// TIA Portal V15.1 export
// export: Created 2024-05-17T05:38:26.0543023Z, ExportSetting WithDefaults, DisplayName Totally Integrated Automation Portal, DisplayVersion V15.1 Update 5, DisplayName TIA Portal Openness, DisplayVersion V15.1 Update 5, DisplayName SINAMICS Startdrive Advanced, DisplayVersion V15.1, DisplayName G130, G150, S120, S150, SINAMICS MV, S210, DisplayVersion V15.1, DisplayName G110M, G120, G120C, G120D, G120P, DisplayVersion V15.1, DisplayName STEP 7 Professional, DisplayVersion V15.1 Update 5, DisplayName STEP 7 Safety, DisplayVersion V15.1, DisplayName WinCC Professional, DisplayVersion V15.1 Update 5, DisplayName SIMATIC Visualization Architect, DisplayVersion V15.1
FUNCTION "LETAFuseName" : Void   // FC2102, SCL
{ S7_Optimized_Access := 'TRUE' }
VERSION : 0.1
// stored: AutoNumber false, IsIECCheckEnabled false, SetENOAutomatically False, UDAEnableTagReadback false
   VAR_INPUT
      I_DBName : String;   // DB Name
      C_Config : "ETAFuseCPC20PNConfig";   // Config / Description About Type Of Object
   END_VAR
   VAR_OUTPUT
      O_FuseNr : Int;   // Fuse number in "STRUCT"
      O_FuseNameOK : Bool;   // Fuse name is found one time by the config
      O_FuseNameNOK : Bool;   // Fuse name is not found by the config or Instance name DB is wrong
      O_FuseNameMoreThenOne : Bool;   // Fuse name is found more then one time by the config
   END_VAR
   VAR_TEMP
      Index : Int;   // Index
      SubIndex : Int;   // Sub Index
   END_VAR
BEGIN
   #Index := 1;
   #SubIndex := 0;

   WHILE (#Index <= 64) DO
       IF (#C_Config.Fuse[#Index].Name = #I_DBName) THEN
           #O_FuseNr := #Index;
           #SubIndex := #SubIndex + 1;
       END_IF;
       #Index := #Index + 1;
   END_WHILE;

   IF (#SubIndex = 1) THEN
       #O_FuseNameOK := True;
       #O_FuseNameNOK := False;
       #O_FuseNameMoreThenOne := False;
   END_IF;

   IF (#SubIndex = 0) THEN
       #O_FuseNameOK := False;
       #O_FuseNameNOK := True;
       #O_FuseNameMoreThenOne := False;
       #O_FuseNr := 0;
   END_IF;

   IF (#SubIndex > 1) THEN
       #O_FuseNameOK := False;
       #O_FuseNameNOK := False;
       #O_FuseNameMoreThenOne := True;
       #O_FuseNr := 0;
   END_IF;
END_FUNCTION
